// TIA Portal V17 export
// export: Created 2025-03-05T08:02:25.2436641Z, ExportSetting WithDefaults, DisplayName Totally Integrated Automation Portal, DisplayVersion V17 Update 8, DisplayName TIA Portal Openness, DisplayVersion V17 Update 8, DisplayName TIA Portal Version Control Interface, DisplayVersion V17, DisplayName SINAMICS Startdrive Advanced, DisplayVersion V17 SP2, DisplayName SINAMICS Startdrive G110M, G120, G120C, G120D, G120P, G115D, DisplayVersion V17 SP2, DisplayName SINAMICS Startdrive G130, G150, S120, S150, SINAMICS MV, S210, DisplayVersion V17 SP2, DisplayName STEP 7 Professional, DisplayVersion V17 Update 8, DisplayName SINUMERIK ONE STEP 7 Toolbox, DisplayVersion V17 Update 12, DisplayName SINUMERIK 840D sl STEP 7 Toolbox, DisplayVersion V17 Update 12, DisplayName STEP 7 Safety, DisplayVersion V17 Update 6, DisplayName WinCC Advanced, DisplayVersion V17 Update 8
TYPE "PART_STATUS_CLADDING"
// stored: IsFailsafeCompliant false
   STRUCT
      STATUS : Struct   // PART STATUS
         PRESENT : Bool;   // PART PRESENT
         OK : Bool;   // PART OK
         PART_REJECTED : Bool;   // PART REJECTED
         QUALITY_PART : Bool;   // PART QUALITY
         FULL_DEPTH : Bool;   // FULL DEPTH / PART FULL DEPTH
         MASTER_PART : Bool;   // MASTER PART / PART MASTER PART
         VIRTUAL_PART : Bool;   // PART VIRTUAL PART
         PART_TYPE : Byte;   // PART TYPE
         PART_MAIN_STATUS_COLOR : Int;   // PART MAIN STATUS HMI COLOR
         PART_CELL_STATUS_COLOR : Int;   // PART CELL STATUS HMI COLOR
         QUALITY_CHECK_STATUS : Struct
            PART_ON_DEMAND : Bool;   // PART QUALITY PART ON DEMAND
            TOOL_CHANGED : Bool;   // PART QUALITY TOOL CHANGED
            PART_TYPE_CHANGED : Bool;   // PART QUALITY PART TYPE CHANGED
            FIRST_CYCLE : Bool;   // PART QUALITY CHECK CYCLE INTERRUMPED
            SPARE : Byte;
         END_STRUCT;
         UNIT_01_STATUS : Struct
            PROCESSED_IN_F1 : Bool;   // PART UNIT 01 PROCESSED IN FIXTURE 1
            PROCESSED_IN_F2 : Bool;   // PART UNIT 01 PROCESSED IN FIXTURE 2
            PROCESSED_IN_F3 : Bool;   // PART UNIT 01 PROCESSED IN FIXTURE 3
            PROCESSED_IN_F4 : Bool;   // PART UNIT 01 PROCESSED IN FIXTURE 4
            FACE_R_STATION_1_DONE : Bool;   // PART UNIT 01 FACE R STATION 1 DONE
            FACE_R_STATION_2_DONE : Bool;   // PART UNIT 01 FACE R STATION 2 DONE
            FACE_R_STATION_3_DONE : Bool;   // PART UNIT 01 FACE R STATION 3 DONE
            FACE_R_STATION_4_DONE : Bool;   // PART UNIT 01 FACE R STATION 4 DONE
            FACE_N_STATION_1_DONE : Bool;   // PART UNIT 01 FACE N STATION 1 DONE
            FACE_N_STATION_2_DONE : Bool;   // PART UNIT 01 FACE N STATION 2 DONE
            FACE_N_STATION_3_DONE : Bool;   // PART UNIT 01 FACE N STATION 3 DONE
            FACE_N_STATION_4_DONE : Bool;   // PART UNIT 01 FACE N STATION 4 DONE
         END_STRUCT;
         UNIT_02_STATUS : Struct
            PROCESSED_IN_F1 : Bool;   // PART UNIT 02 PROCESSED IN FIXTURE 1
            PROCESSED_IN_F2 : Bool;   // PART UNIT 02 PROCESSED IN FIXTURE 2
            PROCESSED_IN_F3 : Bool;   // PART UNIT 02 PROCESSED IN FIXTURE 3
            PROCESSED_IN_F4 : Bool;   // PART UNIT 02 PROCESSED IN FIXTURE 4
            FACE_R_STATION_1_DONE : Bool;   // PART UNIT 02 FACE R STATION 1 DONE
            FACE_R_STATION_2_DONE : Bool;   // PART UNIT 02 FACE R STATION 2 DONE
            FACE_R_STATION_3_DONE : Bool;   // PART UNIT 02 FACE R STATION 3 DONE
            FACE_R_STATION_4_DONE : Bool;   // PART UNIT 02 FACE R STATION 4 DONE
            FACE_N_STATION_1_DONE : Bool;   // PART UNIT 02 FACE N STATION 1 DONE
            FACE_N_STATION_2_DONE : Bool;   // PART UNIT 02 FACE N STATION 2 DONE
            FACE_N_STATION_3_DONE : Bool;   // PART UNIT 02 FACE N STATION 3 DONE
            FACE_N_STATION_4_DONE : Bool;   // PART UNIT 02 FACE N STATION 4 DONE
         END_STRUCT;
         CELL_STATUS : Struct
            NEW : Bool;   // PART NEW
            NEW_CAMARA_OK : Bool;   // PART NEW CAMARA OK
            NEW_IN_TRANSIT : Bool;   // PART NEW IN TRANSIT
            U01_ONE_FACE_DONE : Bool;   // PART UNIT 01 ONE FACE DONE
            U01_ONE_FACE_DONE_ROTATED : Bool;   // PART UNIT 01 ONE FACE DONE ROTATED
            U01_DONE : Bool;   // PART UNIT 01 BOTH FACES DONE
            U01_DONE_IN_TRANSIT : Bool;   // PART UNIT 01 DONE IN TRANSIT
            U02_ONE_FACE_DONE : Bool;   // PART UNIT 02 ONE FACE DONE
            U02_ONE_FACE_DONE_IN_TRANSIT : Bool;   // PART UNIT 02 ONE FACE DONE IN TRANSIT
            U02_ONE_FACE_DONE_ROTATED : Bool;   // PART UNIT 02 ONE FACE DONE ROTATED
            U02_DONE : Bool;   // PART UNIT 02 BOTH FACES DONE
            U02_DONE_IN_TRANSIT : Bool;   // PART UNTI 02 DONE IN TRANSIT
            COOLING_DONE : Bool;   // PART COOLING DONE
            INSPECTION_DONE : Bool;   // PART INSPECTION DONE
            OUTFEED_CAMARA_OK : Bool;   // PART OUTFEED CAMARA OK
            SPARE2 : Bool;
            SPARE3 : Bool;
            SPARE4 : Bool;
            SPARE5 : Bool;
            SPARE6 : Bool;   // PART ROTATION 2 NEW PART
            SPARE7 : Bool;
            SPARE8 : Bool;
            SPARE9 : Bool;
            SPARE10 : Bool;
            SPARE11 : Bool;
            SPARE12 : Bool;
         END_STRUCT;
      END_STRUCT;
      PART_ID : Array[0..99] of Char;   // PART ID
      SPARE : Array[0..10] of Byte;
   END_STRUCT;
END_TYPE
